Yaskawa INFORM job: R2_W27-A6(-180,180).JBI

/JOB
//NAME R2_W27-A6(-180,180)
//POS
///NPOS 27,27,0,2,0,0
///TOOL 0
///POSTYPE PULSE
///PULSE
C00000=92221,-106521,-74255,30348,36888,-11679
C00001=130810,-27044,-38834,46192,102022,-68836
C00002=130792,-26153,-28925,45308,98022,-70722
C00003=133083,-25489,-28460,45385,96895,-70143
C00004=133993,-25185,-28246,45408,96449,-69912
C00005=135092,-24784,-27964,45430,95913,-69634
C00006=133993,-25185,-28246,45408,96449,-69912
C00007=128102,-26791,-29369,51238,107404,-70756
C00008=128116,-26966,-29490,51235,107385,-70758
C00009=128102,-26791,-29369,51238,107404,-70756
C00010=132266,-25772,-28984,36275,85586,-70414
C00011=140457,-22353,-26557,35352,82376,-68071
C00012=140457,-22303,-26199,35364,82216,-68122
C00013=140457,-22353,-26557,35352,82376,-68071
C00014=137889,-28846,-36558,35564,85755,-68039
C00015=120712,-3842,-12080,46489,110386,42187
C00016=120713,-3846,-12083,46489,110386,42187
C00017=120002,-4638,-12864,46405,110804,42030
C00018=120716,-5911,-13493,46430,110248,42119
C00019=120713,-4021,-13473,46730,110921,42463
C00020=122947,-4573,-12811,46825,109275,42782
C00021=120713,-3830,-12070,46489,110386,42187
C00022=120712,-3826,-12067,46489,110386,42187
C00023=124791,-46459,-52790,31112,79590,55440
C00024=127667,-74453,-59286,20057,47641,61356
C00025=74334,-163397,-127461,41990,65126,41829
C00026=74334,-163397,-127461,41990,65126,41829
BC00000=394390,175993,1075172
BC00001=398174,104699,1075175
BC00002=398174,104704,1027742
BC00003=398174,108892,1013252
BC00004=398174,110567,1007456
BC00005=398174,110557,1007452
BC00006=398174,110567,1007456
BC00007=398174,95671,973938
BC00008=398174,98743,973937
BC00009=398174,95671,973938
BC00010=398174,135761,1075175
BC00011=398174,139769,1075175
BC00012=398174,139769,1066495
BC00013=398174,139769,1075175
BC00014=398174,135761,1075175
BC00015=361280,141408,1067859
BC00016=358550,143625,1043827
BC00017=357489,144487,1034483
BC00018=357458,144512,1034214
BC00019=357458,144512,1034214
BC00020=357489,144487,1034483
BC00021=353135,143604,1043818
BC00022=355865,141386,1067851
BC00023=355865,141386,1067851
BC00024=355865,141386,1067851
BC00025=355865,141386,1067851
BC00026=269302,274694,1067851
///POSTYPE BASE
///RECTAN
///RCONF 0,0,0,0,1,0,0,0,0,0,0,0,0,0,0,0,0,0,0,0,0,0,0,0
P00001=1521.784,432.249,299.876,0.4361,26.2594,39.1916
P00006=2.006,1.622,-0.565,0.0000,0.0000,0.0000
//INST
///DATE 2023/11/09 19:26
///ATTR SC,RW
///GROUP1 RB1,BS1
NOP
'r2_W27-A6(-180,180)
'
'Path S852
SFTOF
MOVJ C00000 BC00000 VJ=25.00
MOVJ C00001 BC00001 VJ=100.00
MOVJ C00002 BC00002 VJ=100.00
MOVL C00003 BC00003 V=400.0
MOVL C00004 BC00004 V=60.0
REFP 3 C00005 BC00005
CALL JOB:SEARCH-R1
SET P001 P006
SFTON P001
MOVL C00006 BC00006 V=60.0
MOVL C00007 BC00007 V=60.0
REFP 3 C00008 BC00008
CALL JOB:SEARCH-R1
SET P001 P006
SFTON P001
MOVL C00009 BC00009 V=60.0
MOVL C00010 BC00010 V=100.0
MOVL C00011 BC00011 V=60.0
REFP 3 C00012 BC00012
CALL JOB:SEARCH-R1
SET P001 P006
SFTON P001
MOVL C00013 BC00013 V=60.0
MOVL C00014 BC00014 V=100.0
'Path W853
SFTOF
SFTON P001
MOVJ C00015 BC00015 VJ=100.00
MOVL C00016 BC00016 V=400.0
MOVL C00017 BC00017 V=100.0 PL=0
REFP 1 C00018 BC00018
REFP 2 C00019 BC00019
MACRO1 MJ#(0) ARGF0
ARCON
MOVL C00020 BC00020 V=10.0
ARCOF
MOVL C00021 BC00021 V=400.0
MOVL C00022 BC00022 V=1000.0
SFTOF
MOVJ C00023 BC00023 VJ=25.00
MOVJ C00024 BC00024 VJ=25.00
MOVJ C00025 BC00025 VJ=25.00
MOVJ C00026 BC00026 VJ=25.00
END
